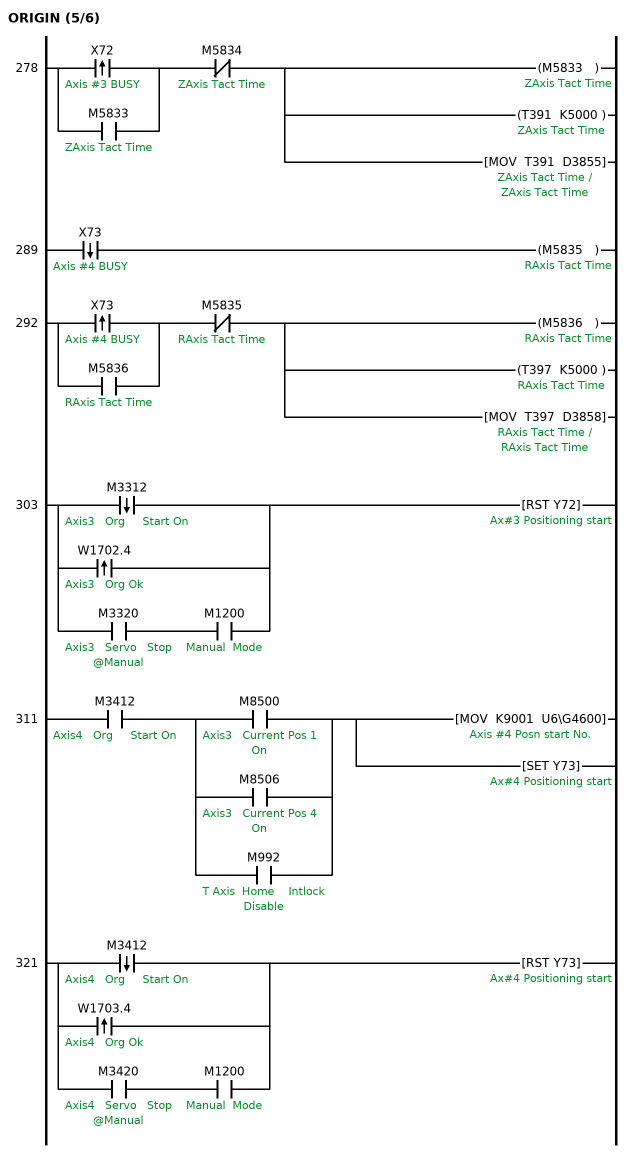
[picture p24: ladder of ORIGIN, rungs at steps 278 to 321]
278   LDP     X72  ; Axis #3 BUSY
      OR      M5833  ; ZAxis Tact Time
      ANI     M5834  ; ZAxis Tact Time
      OUT     M5833  ; ZAxis Tact Time
      OUT     T391 K5000  ; ZAxis Tact Time
      MOV     T391 D3855  ; ZAxis Tact Time
289   LDF     X73  ; Axis #4 BUSY
      OUT     M5835  ; RAxis Tact Time
292   LDP     X73  ; Axis #4 BUSY
      OR      M5836  ; RAxis Tact Time
      ANI     M5835  ; RAxis Tact Time
      OUT     M5836  ; RAxis Tact Time
      OUT     T397 K5000  ; RAxis Tact Time
      MOV     T397 D3858  ; RAxis Tact Time
303   LDF     M3312  ; Axis3   Org     Start On
      ORP     W1702.4  ; Axis3   Org Ok
      LD      M3320  ; Axis3   Servo   Stop    @Manual
      AND     M1200  ; Manual  Mode
      ORB
      RST     Y72  ; Ax#3 Positioning start
311   LD      M3412  ; Axis4   Org     Start On
      LD      M8500  ; Axis3   Current Pos 1 On
      OR      M8506  ; Axis3   Current Pos 4 On
      OR      M992  ; T Axis  Home    Intlock Disable
      ANB
      MOV     K9001 U6\G4600  ; Axis #4 Posn start No.
      SET     Y73  ; Ax#4 Positioning start
321   LDF     M3412  ; Axis4   Org     Start On
      ORP     W1703.4  ; Axis4   Org Ok
      LD      M3420  ; Axis4   Servo   Stop    @Manual
      AND     M1200  ; Manual  Mode
      ORB
      RST     Y73  ; Ax#4 Positioning start
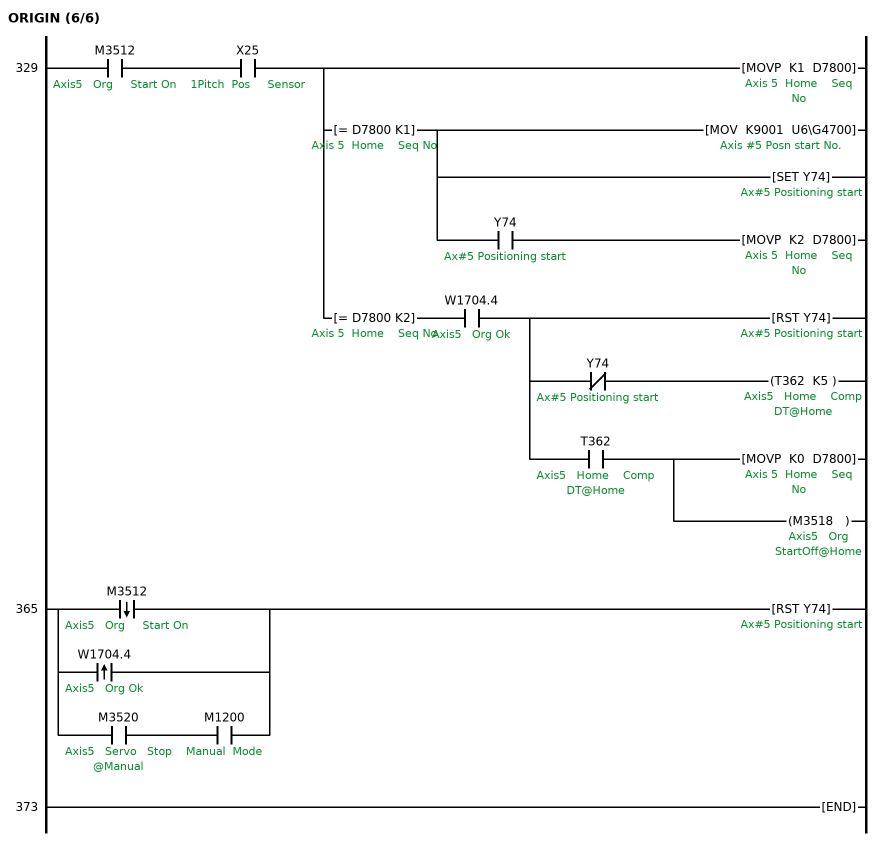
329   LD      M3512  ; Axis5   Org     Start On
      AND     X25  ; 1Pitch  Pos     Sensor
      MOVP    K1 D7800  ; Axis 5  Home    Seq No
      MPS
      AND=    D7800 K1  ; Axis 5  Home    Seq No
      MOV     K9001 U6\G4700  ; Axis #5 Posn start No.
      SET     Y74  ; Ax#5 Positioning start
      AND     Y74  ; Ax#5 Positioning start
      MOVP    K2 D7800
      MPP
      AND=    D7800 K2  ; Axis 5  Home    Seq No
      AND     W1704.4  ; Axis5   Org Ok
      RST     Y74  ; Ax#5 Positioning start
      MPS
      ANI     Y74  ; Ax#5 Positioning start
      OUT     T362 K5  ; Axis5   Home    Comp    DT@Home
      MPP
      AND     T362  ; Axis5   Home    Comp    DT@Home
      MOVP    K0 D7800
      OUT     M3518  ; Axis5   Org     StartOff@Home
365   LDF     M3512  ; Axis5   Org     Start On
      ORP     W1704.4  ; Axis5   Org Ok
      LD      M3520  ; Axis5   Servo   Stop    @Manual
      AND     M1200  ; Manual  Mode
      ORB
      RST     Y74  ; Ax#5 Positioning start
373   END
END_PROGRAM

PROGRAM ALARM
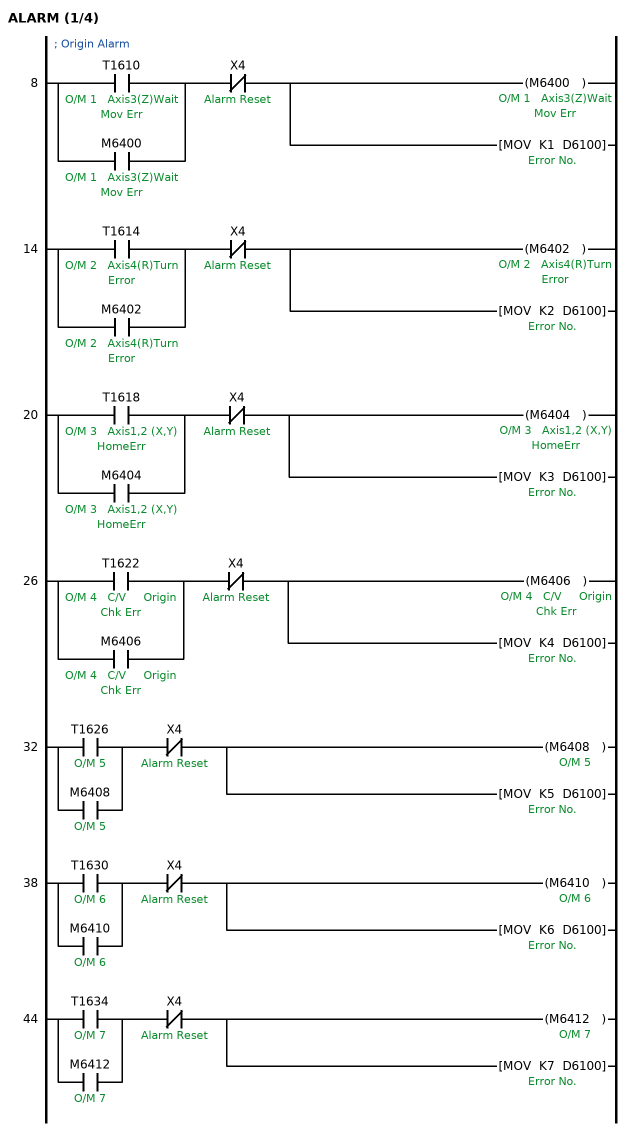
; Origin Alarm
8     LD      T1610  ; O/M 1   Axis3(Z)Wait    Mov Err
      OR      M6400  ; O/M 1   Axis3(Z)Wait    Mov Err
      ANI     X4  ; Alarm Reset
      OUT     M6400  ; O/M 1   Axis3(Z)Wait    Mov Err
      MOV     K1 D6100  ; Error No.
14    LD      T1614  ; O/M 2   Axis4(R)Turn    Error
      OR      M6402  ; O/M 2   Axis4(R)Turn    Error
      ANI     X4  ; Alarm Reset
      OUT     M6402  ; O/M 2   Axis4(R)Turn    Error
      MOV     K2 D6100
20    LD      T1618  ; O/M 3   Axis1,2 (X,Y)   HomeErr
      OR      M6404  ; O/M 3   Axis1,2 (X,Y)   HomeErr
      ANI     X4  ; Alarm Reset
      OUT     M6404  ; O/M 3   Axis1,2 (X,Y)   HomeErr
      MOV     K3 D6100
26    LD      T1622  ; O/M 4   C/V     Origin  Chk Err
      OR      M6406  ; O/M 4   C/V     Origin  Chk Err
      ANI     X4  ; Alarm Reset
      OUT     M6406  ; O/M 4   C/V     Origin  Chk Err
      MOV     K4 D6100
32    LD      T1626  ; O/M 5
      OR      M6408  ; O/M 5
      ANI     X4  ; Alarm Reset
      OUT     M6408  ; O/M 5
      MOV     K5 D6100
38    LD      T1630  ; O/M 6
      OR      M6410  ; O/M 6
      ANI     X4  ; Alarm Reset
      OUT     M6410  ; O/M 6
      MOV     K6 D6100
44    LD      T1634  ; O/M 7
      OR      M6412  ; O/M 7
      ANI     X4  ; Alarm Reset
      OUT     M6412  ; O/M 7
      MOV     K7 D6100
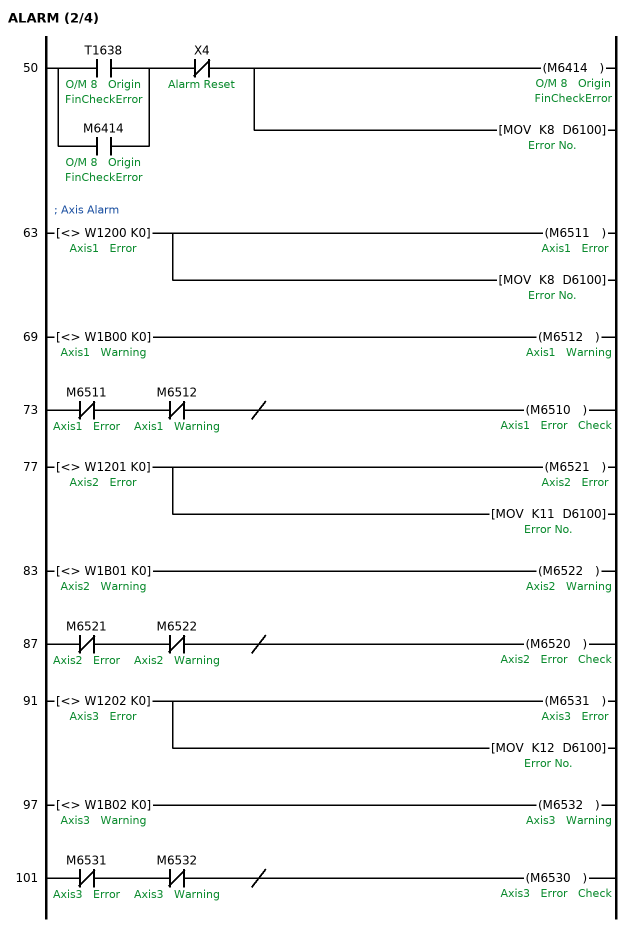
50    LD      T1638  ; O/M 8   Origin  FinCheckError
      OR      M6414  ; O/M 8   Origin  FinCheckError
      ANI     X4  ; Alarm Reset
      OUT     M6414  ; O/M 8   Origin  FinCheckError
      MOV     K8 D6100
; Axis Alarm
63    LD<>    W1200 K0  ; Axis1   Error
      OUT     M6511  ; Axis1   Error
      MOV     K8 D6100
69    LD<>    W1B00 K0  ; Axis1   Warning
      OUT     M6512  ; Axis1   Warning
73    LDI     M6511  ; Axis1   Error
      ANI     M6512  ; Axis1   Warning
      INV
      OUT     M6510  ; Axis1   Error   Check
77    LD<>    W1201 K0  ; Axis2   Error
      OUT     M6521  ; Axis2   Error
      MOV     K11 D6100
83    LD<>    W1B01 K0  ; Axis2   Warning
      OUT     M6522  ; Axis2   Warning
87    LDI     M6521  ; Axis2   Error
      ANI     M6522  ; Axis2   Warning
      INV
      OUT     M6520  ; Axis2   Error   Check
91    LD<>    W1202 K0  ; Axis3   Error
      OUT     M6531  ; Axis3   Error
      MOV     K12 D6100
97    LD<>    W1B02 K0  ; Axis3   Warning
      OUT     M6532  ; Axis3   Warning
101   LDI     M6531  ; Axis3   Error
      ANI     M6532  ; Axis3   Warning
      INV
      OUT     M6530  ; Axis3   Error   Check
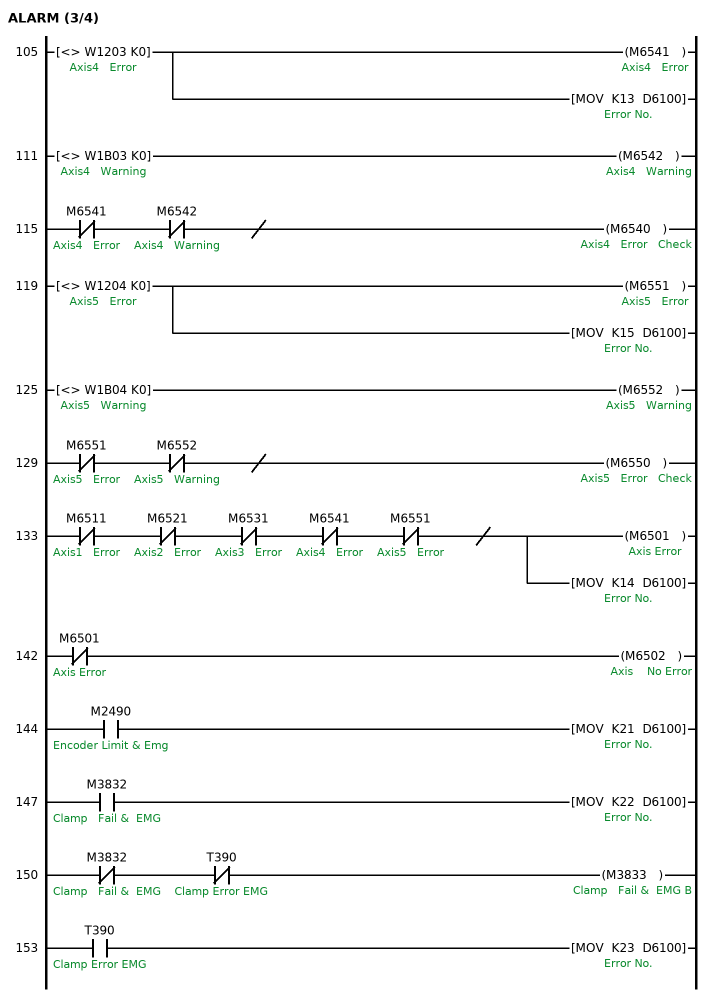
105   LD<>    W1203 K0  ; Axis4   Error
      OUT     M6541  ; Axis4   Error
      MOV     K13 D6100
111   LD<>    W1B03 K0  ; Axis4   Warning
      OUT     M6542  ; Axis4   Warning
115   LDI     M6541  ; Axis4   Error
      ANI     M6542  ; Axis4   Warning
      INV
      OUT     M6540  ; Axis4   Error   Check
119   LD<>    W1204 K0  ; Axis5   Error
      OUT     M6551  ; Axis5   Error
      MOV     K15 D6100
125   LD<>    W1B04 K0  ; Axis5   Warning
      OUT     M6552  ; Axis5   Warning
129   LDI     M6551  ; Axis5   Error
      ANI     M6552  ; Axis5   Warning
      INV
      OUT     M6550  ; Axis5   Error   Check
133   LDI     M6511  ; Axis1   Error
      ANI     M6521  ; Axis2   Error
      ANI     M6531  ; Axis3   Error
      ANI     M6541  ; Axis4   Error
      ANI     M6551  ; Axis5   Error
      INV
      OUT     M6501  ; Axis Error
      MOV     K14 D6100
142   LDI     M6501  ; Axis Error
      OUT     M6502  ; Axis    No Error
144   LD      M2490  ; Encoder Limit & Emg
      MOV     K21 D6100
147   LD      M3832  ; Clamp   Fail &  EMG
      MOV     K22 D6100
150   LDI     M3832  ; Clamp   Fail &  EMG
      ANI     T390  ; Clamp Error EMG
      OUT     M3833  ; Clamp   Fail &  EMG B
153   LD      T390  ; Clamp Error EMG
      MOV     K23 D6100
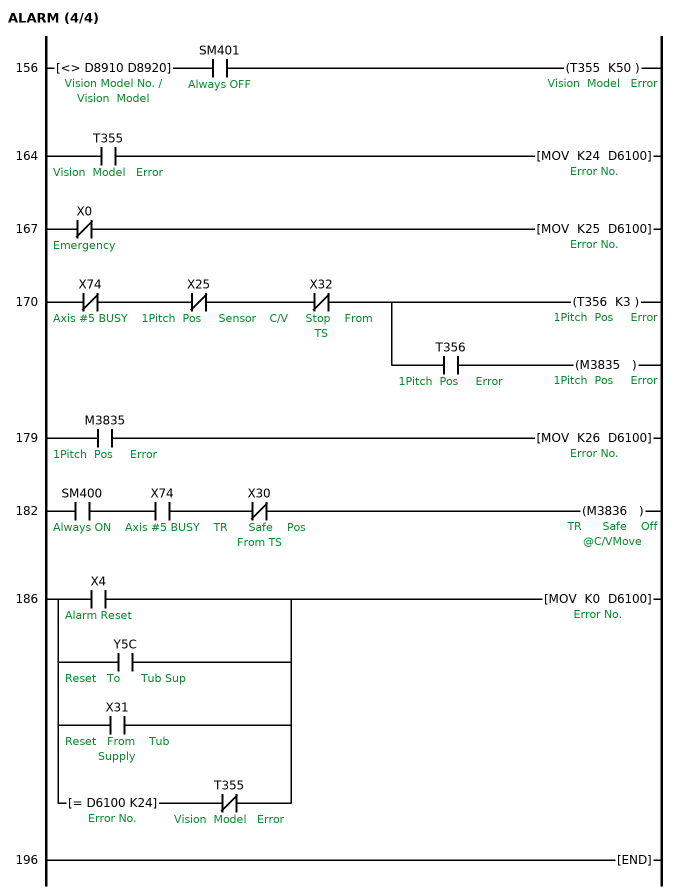
156   LD<>    D8910 D8920  ; Vision Model No. / Vision  Model
      AND     SM401  ; Always OFF
      OUT     T355 K50  ; Vision  Model   Error
164   LD      T355  ; Vision  Model   Error
      MOV     K24 D6100
167   LDI     X0  ; Emergency
      MOV     K25 D6100
170   LDI     X74  ; Axis #5 BUSY
      ANI     X25  ; 1Pitch  Pos     Sensor
      ANI     X32  ; C/V     Stop    From    TS
      OUT     T356 K3  ; 1Pitch  Pos     Error
      AND     T356  ; 1Pitch  Pos     Error
      OUT     M3835  ; 1Pitch  Pos     Error
179   LD      M3835  ; 1Pitch  Pos     Error
      MOV     K26 D6100
182   LD      SM400  ; Always ON
      AND     X74  ; Axis #5 BUSY
      ANI     X30  ; TR      Safe    Pos     From TS
      OUT     M3836  ; TR      Safe    Off     @C/VMove
186   LD      X4  ; Alarm Reset
      OR      Y5C  ; Reset   To      Tub Sup
      OR      X31  ; Reset   From    Tub     Supply
      LD=     D6100 K24  ; Error No.
      ANI     T355  ; Vision  Model   Error
      ORB
      MOV     K0 D6100
196   END
END_PROGRAM

PROGRAM SERVO
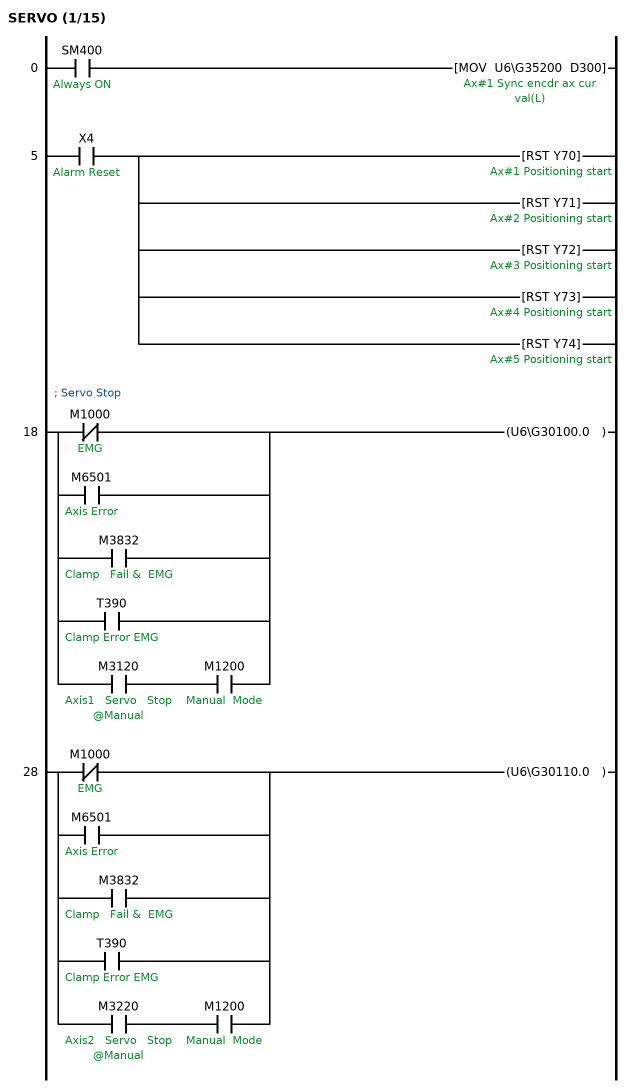
0     LD      SM400  ; Always ON
      MOV     U6\G35200 D300  ; Ax#1 Sync encdr ax cur val(L)
5     LD      X4  ; Alarm Reset
      RST     Y70  ; Ax#1 Positioning start
      RST     Y71  ; Ax#2 Positioning start
      RST     Y72  ; Ax#3 Positioning start
      RST     Y73  ; Ax#4 Positioning start
      RST     Y74  ; Ax#5 Positioning start
; Servo Stop
18    LDI     M1000  ; EMG
      OR      M6501  ; Axis Error
      OR      M3832  ; Clamp   Fail &  EMG
      OR      T390  ; Clamp Error EMG
      LD      M3120  ; Axis1   Servo   Stop    @Manual
      AND     M1200  ; Manual  Mode
      ORB
      OUT     U6\G30100.0
28    LDI     M1000  ; EMG
      OR      M6501  ; Axis Error
      OR      M3832  ; Clamp   Fail &  EMG
      OR      T390  ; Clamp Error EMG
      LD      M3220  ; Axis2   Servo   Stop    @Manual
      AND     M1200  ; Manual  Mode
      ORB
      OUT     U6\G30110.0
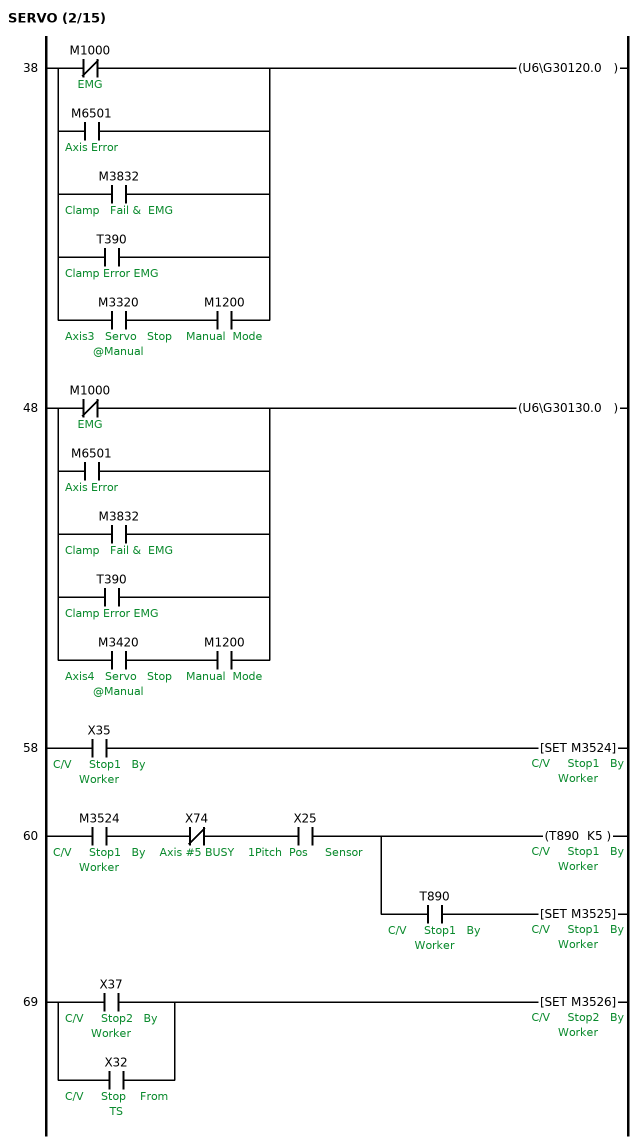
38    LDI     M1000  ; EMG
      OR      M6501  ; Axis Error
      OR      M3832  ; Clamp   Fail &  EMG
      OR      T390  ; Clamp Error EMG
      LD      M3320  ; Axis3   Servo   Stop    @Manual
      AND     M1200  ; Manual  Mode
      ORB
      OUT     U6\G30120.0
48    LDI     M1000  ; EMG
      OR      M6501  ; Axis Error
      OR      M3832  ; Clamp   Fail &  EMG
      OR      T390  ; Clamp Error EMG
      LD      M3420  ; Axis4   Servo   Stop    @Manual
      AND     M1200  ; Manual  Mode
      ORB
      OUT     U6\G30130.0
58    LD      X35  ; C/V     Stop1   By      Worker
      SET     M3524  ; C/V     Stop1   By      Worker
60    LD      M3524  ; C/V     Stop1   By      Worker
      ANI     X74  ; Axis #5 BUSY
      AND     X25  ; 1Pitch  Pos     Sensor
      OUT     T890 K5  ; C/V     Stop1   By      Worker
      AND     T890  ; C/V     Stop1   By      Worker
      SET     M3525  ; C/V     Stop1   By      Worker
69    LD      X37  ; C/V     Stop2   By      Worker
      OR      X32  ; C/V     Stop    From    TS
      SET     M3526  ; C/V     Stop2   By      Worker
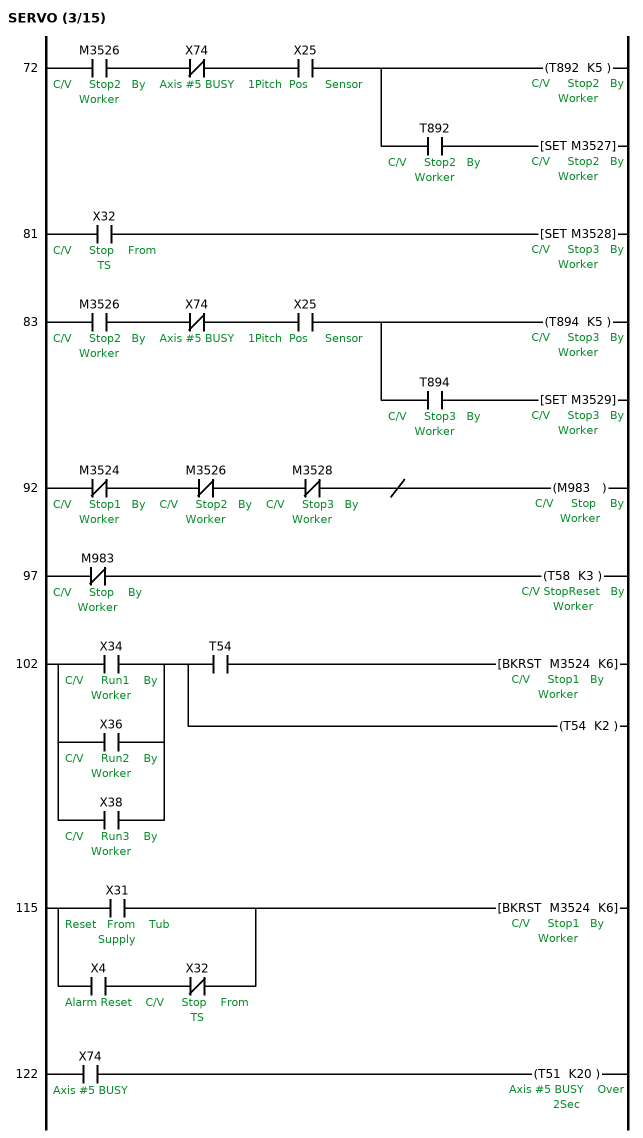
72    LD      M3526  ; C/V     Stop2   By      Worker
      ANI     X74  ; Axis #5 BUSY
      AND     X25  ; 1Pitch  Pos     Sensor
      OUT     T892 K5  ; C/V     Stop2   By      Worker
      AND     T892  ; C/V     Stop2   By      Worker
      SET     M3527  ; C/V     Stop2   By      Worker
81    LD      X32  ; C/V     Stop    From    TS
      SET     M3528  ; C/V     Stop3   By      Worker
83    LD      M3526  ; C/V     Stop2   By      Worker
      ANI     X74  ; Axis #5 BUSY
      AND     X25  ; 1Pitch  Pos     Sensor
      OUT     T894 K5  ; C/V     Stop3   By      Worker
      AND     T894  ; C/V     Stop3   By      Worker
      SET     M3529  ; C/V     Stop3   By      Worker
92    LDI     M3524  ; C/V     Stop1   By      Worker
      ANI     M3526  ; C/V     Stop2   By      Worker
      ANI     M3528  ; C/V     Stop3   By      Worker
      INV
      OUT     M983  ; C/V     Stop    By      Worker
97    LDI     M983  ; C/V     Stop    By      Worker
      OUT     T58 K3  ; C/V StopReset   By      Worker
102   LD      X34  ; C/V     Run1    By      Worker
      OR      X36  ; C/V     Run2    By      Worker
      OR      X38  ; C/V     Run3    By      Worker
      MPS
      AND     T54
      BKRST   M3524 K6
      MPP
      OUT     T54 K2
115   LD      X31  ; Reset   From    Tub     Supply
      LD      X4  ; Alarm Reset
      ANI     X32  ; C/V     Stop    From    TS
      ORB
      BKRST   M3524 K6
122   LD      X74  ; Axis #5 BUSY
      OUT     T51 K20  ; Axis #5 BUSY    Over    2Sec
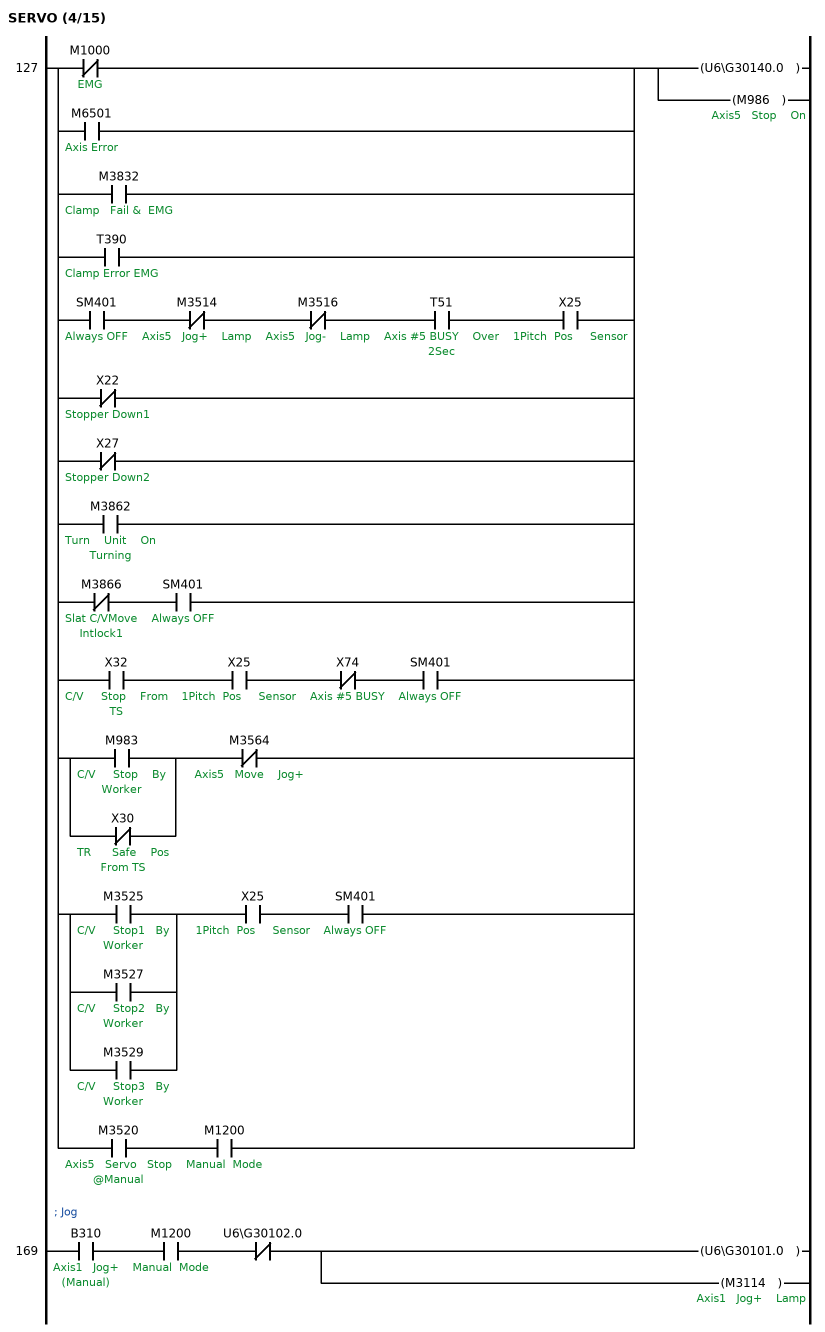
127   LDI     M1000  ; EMG
      OR      M6501  ; Axis Error
      OR      M3832  ; Clamp   Fail &  EMG
      OR      T390  ; Clamp Error EMG
      LD      SM401  ; Always OFF
      ANI     M3514  ; Axis5   Jog+    Lamp
      ANI     M3516  ; Axis5   Jog-    Lamp
      AND     T51  ; Axis #5 BUSY    Over    2Sec
      AND     X25  ; 1Pitch  Pos     Sensor
      ORB
      ORI     X22  ; Stopper Down1
      ORI     X27  ; Stopper Down2
      OR      M3862  ; Turn    Unit    On      Turning
      LDI     M3866  ; Slat C/VMove    Intlock1
      AND     SM401  ; Always OFF
      ORB
      LD      X32  ; C/V     Stop    From    TS
      AND     X25  ; 1Pitch  Pos     Sensor
      ANI     X74  ; Axis #5 BUSY
      AND     SM401  ; Always OFF
      ORB
      LD      M983  ; C/V     Stop    By      Worker
      ORI     X30  ; TR      Safe    Pos     From TS
      ANI     M3564  ; Axis5   Move    Jog+
      ORB
      LD      M3525  ; C/V     Stop1   By      Worker
      OR      M3527  ; C/V     Stop2   By      Worker
      OR      M3529  ; C/V     Stop3   By      Worker
      AND     X25  ; 1Pitch  Pos     Sensor
      AND     SM401  ; Always OFF
      ORB
      LD      M3520  ; Axis5   Servo   Stop    @Manual
      AND     M1200  ; Manual  Mode
      ORB
      OUT     U6\G30140.0
      OUT     M986  ; Axis5   Stop    On
; Jog
169   LD      B310  ; Axis1   Jog+    (Manual)
      AND     M1200  ; Manual  Mode
      ANI     U6\G30102.0
      OUT     U6\G30101.0
      OUT     M3114  ; Axis1   Jog+    Lamp
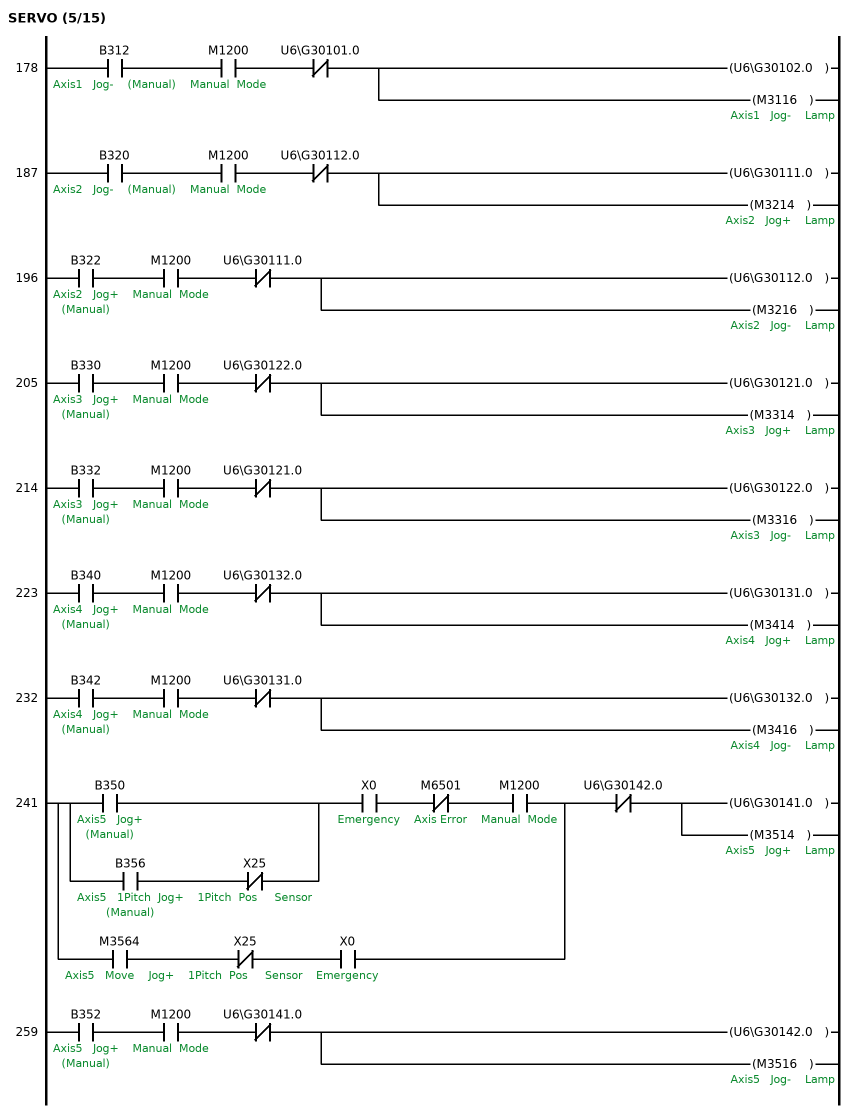
178   LD      B312  ; Axis1   Jog-    (Manual)
      AND     M1200  ; Manual  Mode
      ANI     U6\G30101.0
      OUT     U6\G30102.0
      OUT     M3116  ; Axis1   Jog-    Lamp
187   LD      B320  ; Axis2   Jog-    (Manual)
      AND     M1200  ; Manual  Mode
      ANI     U6\G30112.0
      OUT     U6\G30111.0
      OUT     M3214  ; Axis2   Jog+    Lamp
196   LD      B322  ; Axis2   Jog+    (Manual)
      AND     M1200  ; Manual  Mode
      ANI     U6\G30111.0
      OUT     U6\G30112.0
      OUT     M3216  ; Axis2   Jog-    Lamp
205   LD      B330  ; Axis3   Jog+    (Manual)
      AND     M1200  ; Manual  Mode
      ANI     U6\G30122.0
      OUT     U6\G30121.0
      OUT     M3314  ; Axis3   Jog+    Lamp
214   LD      B332  ; Axis3   Jog+    (Manual)
      AND     M1200  ; Manual  Mode
      ANI     U6\G30121.0
      OUT     U6\G30122.0
      OUT     M3316  ; Axis3   Jog-    Lamp
223   LD      B340  ; Axis4   Jog+    (Manual)
      AND     M1200  ; Manual  Mode
      ANI     U6\G30132.0
      OUT     U6\G30131.0
      OUT     M3414  ; Axis4   Jog+    Lamp
232   LD      B342  ; Axis4   Jog+    (Manual)
      AND     M1200  ; Manual  Mode
      ANI     U6\G30131.0
      OUT     U6\G30132.0
      OUT     M3416  ; Axis4   Jog-    Lamp
241   LD      B350  ; Axis5   Jog+    (Manual)
      LD      B356  ; Axis5   1Pitch  Jog+    (Manual)
      ANI     X25  ; 1Pitch  Pos     Sensor
      ORB
      AND     X0  ; Emergency
      ANI     M6501  ; Axis Error
      AND     M1200  ; Manual  Mode
      LD      M3564  ; Axis5   Move    Jog+
      ANI     X25  ; 1Pitch  Pos     Sensor
      AND     X0  ; Emergency
      ORB
      ANI     U6\G30142.0
      OUT     U6\G30141.0
      OUT     M3514  ; Axis5   Jog+    Lamp
259   LD      B352  ; Axis5   Jog+    (Manual)
      AND     M1200  ; Manual  Mode
      ANI     U6\G30141.0
      OUT     U6\G30142.0
      OUT     M3516  ; Axis5   Jog-    Lamp
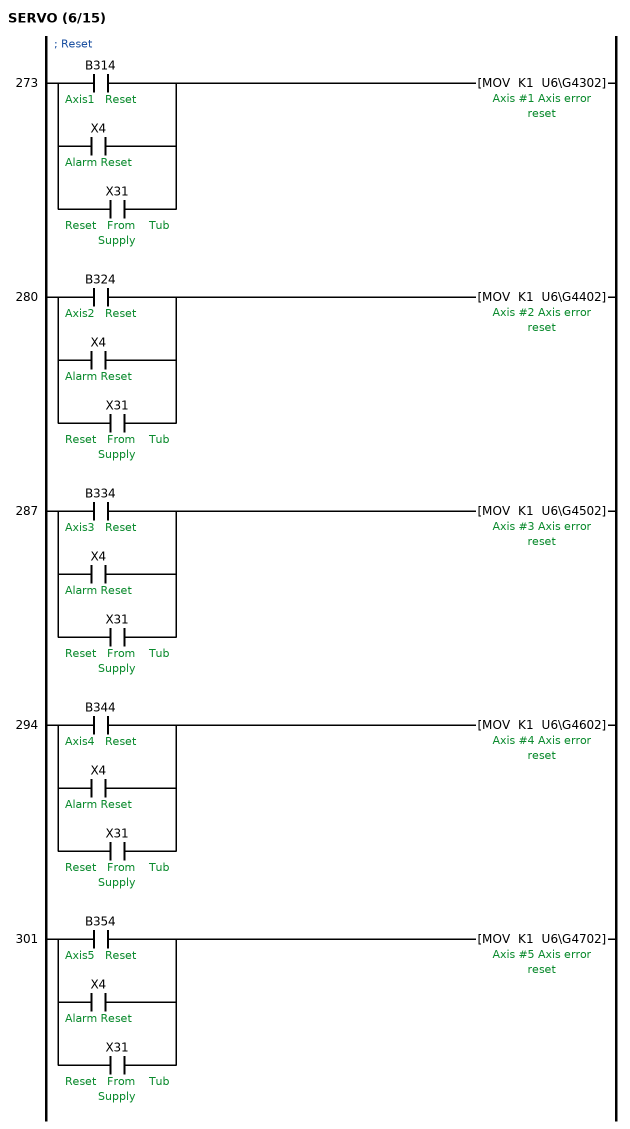
; Reset
273   LD      B314  ; Axis1   Reset
      OR      X4  ; Alarm Reset
      OR      X31  ; Reset   From    Tub     Supply
      MOV     K1 U6\G4302  ; Axis #1 Axis error reset
280   LD      B324  ; Axis2   Reset
      OR      X4  ; Alarm Reset
      OR      X31  ; Reset   From    Tub     Supply
      MOV     K1 U6\G4402  ; Axis #2 Axis error reset
287   LD      B334  ; Axis3   Reset
      OR      X4  ; Alarm Reset
      OR      X31  ; Reset   From    Tub     Supply
      MOV     K1 U6\G4502  ; Axis #3 Axis error reset
294   LD      B344  ; Axis4   Reset
      OR      X4  ; Alarm Reset
      OR      X31  ; Reset   From    Tub     Supply
      MOV     K1 U6\G4602  ; Axis #4 Axis error reset
301   LD      B354  ; Axis5   Reset
      OR      X4  ; Alarm Reset
      OR      X31  ; Reset   From    Tub     Supply
      MOV     K1 U6\G4702  ; Axis #5 Axis error reset
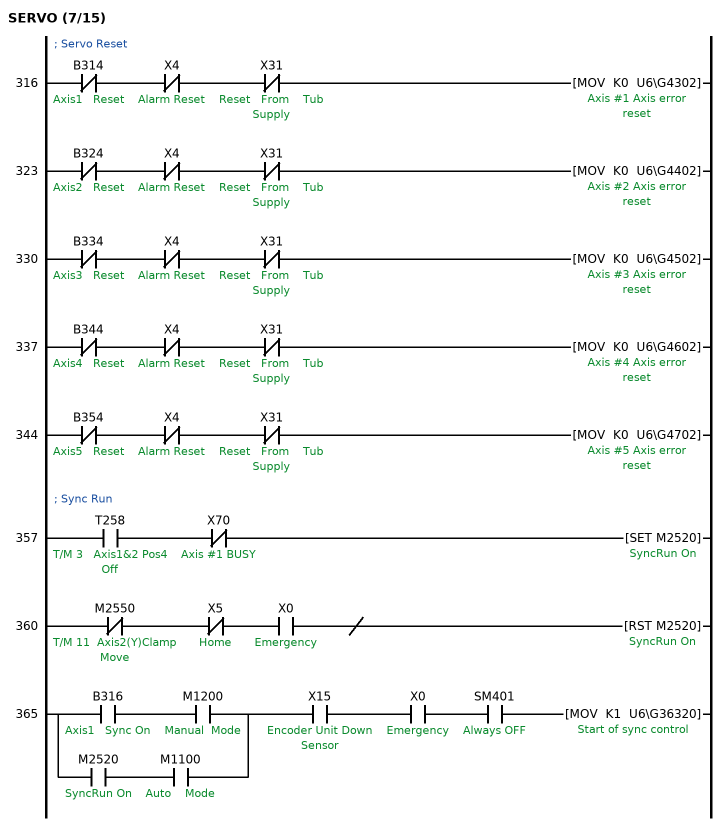
; Servo Reset
316   LDI     B314  ; Axis1   Reset
      ANI     X4  ; Alarm Reset
      ANI     X31  ; Reset   From    Tub     Supply
      MOV     K0 U6\G4302
323   LDI     B324  ; Axis2   Reset
      ANI     X4  ; Alarm Reset
      ANI     X31  ; Reset   From    Tub     Supply
      MOV     K0 U6\G4402
330   LDI     B334  ; Axis3   Reset
      ANI     X4  ; Alarm Reset
      ANI     X31  ; Reset   From    Tub     Supply
      MOV     K0 U6\G4502
337   LDI     B344  ; Axis4   Reset
      ANI     X4  ; Alarm Reset
      ANI     X31  ; Reset   From    Tub     Supply
      MOV     K0 U6\G4602
344   LDI     B354  ; Axis5   Reset
      ANI     X4  ; Alarm Reset
      ANI     X31  ; Reset   From    Tub     Supply
      MOV     K0 U6\G4702
; Sync Run
357   LD      T258  ; T/M 3   Axis1&2 Pos4    Off
      ANI     X70  ; Axis #1 BUSY
      SET     M2520  ; SyncRun On
360   LDI     M2550  ; T/M 11  Axis2(Y)Clamp   Move
      ANI     X5  ; Home
      AND     X0  ; Emergency
      INV
      RST     M2520  ; SyncRun On
365   LD      B316  ; Axis1   Sync On
      AND     M1200  ; Manual  Mode
      LD      M2520  ; SyncRun On
      AND     M1100  ; Auto    Mode
      ORB
      AND     X15  ; Encoder Unit Down Sensor
      AND     X0  ; Emergency
      AND     SM401  ; Always OFF
      MOV     K1 U6\G36320  ; Start of sync control
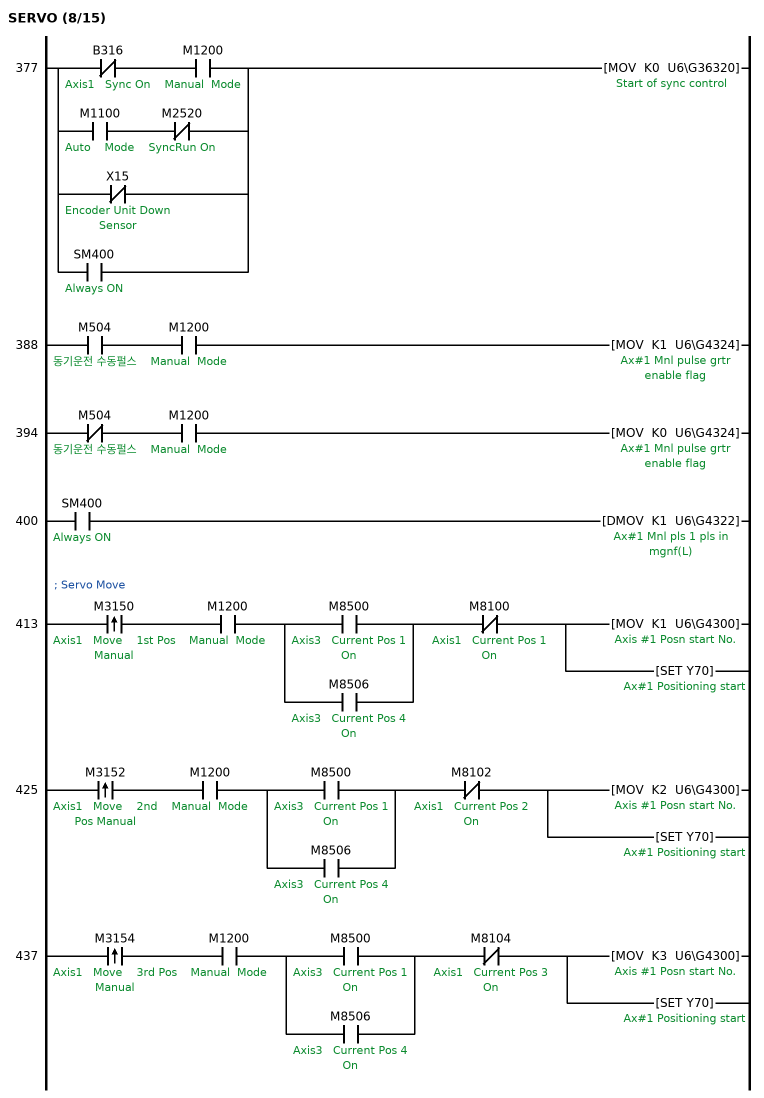
377   LDI     B316  ; Axis1   Sync On
      AND     M1200  ; Manual  Mode
      LD      M1100  ; Auto    Mode
      ANI     M2520  ; SyncRun On
      ORB
      ORI     X15  ; Encoder Unit Down Sensor
      OR      SM400  ; Always ON
      MOV     K0 U6\G36320
388   LD      M504  ; 동기운전 수동펄스
      AND     M1200  ; Manual  Mode
      MOV     K1 U6\G4324  ; Ax#1 Mnl pulse grtr enable flag
394   LDI     M504  ; 동기운전 수동펄스
      AND     M1200  ; Manual  Mode
      MOV     K0 U6\G4324
400   LD      SM400  ; Always ON
      DMOV    K1 U6\G4322  ; Ax#1 Mnl pls 1 pls in mgnf(L)
; Servo Move
413   LDP     M3150  ; Axis1   Move    1st Pos Manual
      AND     M1200  ; Manual  Mode
      LD      M8500  ; Axis3   Current Pos 1 On
      OR      M8506  ; Axis3   Current Pos 4 On
      ANB
      ANI     M8100  ; Axis1   Current Pos 1 On
      MOV     K1 U6\G4300  ; Axis #1 Posn start No.
      SET     Y70  ; Ax#1 Positioning start
425   LDP     M3152  ; Axis1   Move    2nd Pos Manual
      AND     M1200  ; Manual  Mode
      LD      M8500  ; Axis3   Current Pos 1 On
      OR      M8506  ; Axis3   Current Pos 4 On
      ANB
      ANI     M8102  ; Axis1   Current Pos 2 On
      MOV     K2 U6\G4300
      SET     Y70  ; Ax#1 Positioning start
437   LDP     M3154  ; Axis1   Move    3rd Pos Manual
      AND     M1200  ; Manual  Mode
      LD      M8500  ; Axis3   Current Pos 1 On
      OR      M8506  ; Axis3   Current Pos 4 On
      ANB
      ANI     M8104  ; Axis1   Current Pos 3 On
      MOV     K3 U6\G4300
      SET     Y70  ; Ax#1 Positioning start
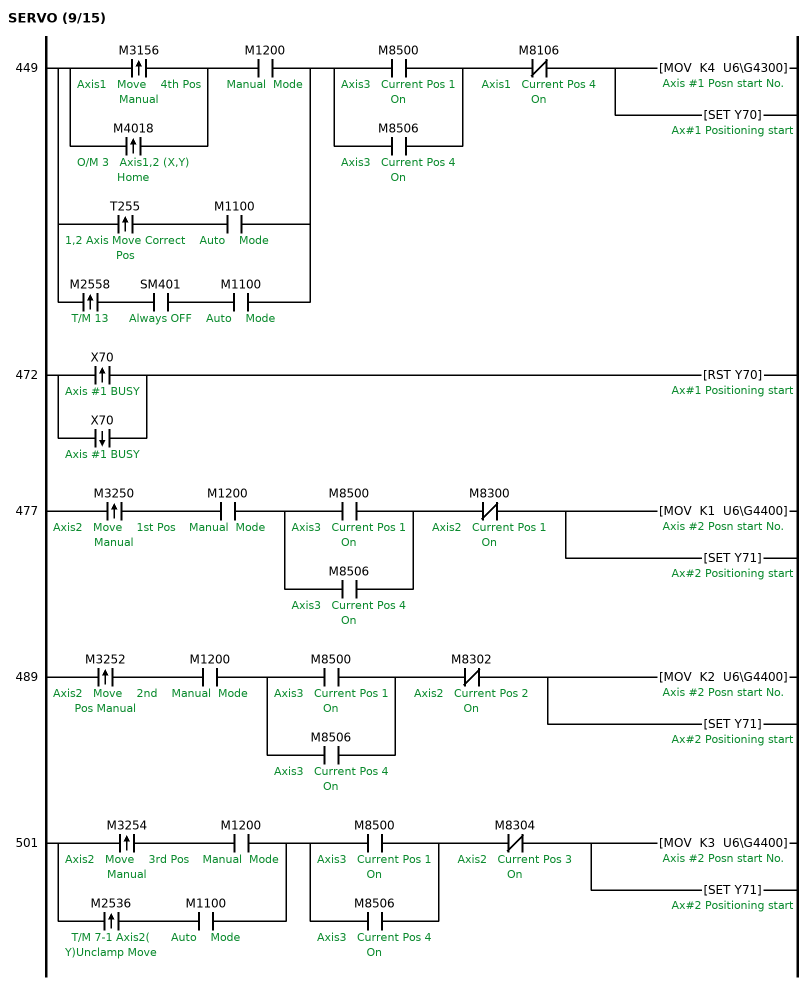
449   LDP     M3156  ; Axis1   Move    4th Pos Manual
      ORP     M4018  ; O/M 3   Axis1,2 (X,Y)   Home
      AND     M1200  ; Manual  Mode
      LDP     T255  ; 1,2 Axis Move Correct Pos
      AND     M1100  ; Auto    Mode
      ORB
      LDP     M2558  ; T/M 13
      AND     SM401  ; Always OFF
      AND     M1100  ; Auto    Mode
      ORB
      LD      M8500  ; Axis3   Current Pos 1 On
      OR      M8506  ; Axis3   Current Pos 4 On
      ANB
      ANI     M8106  ; Axis1   Current Pos 4 On
      MOV     K4 U6\G4300
      SET     Y70  ; Ax#1 Positioning start
472   LDP     X70  ; Axis #1 BUSY
      ORF     X70  ; Axis #1 BUSY
      RST     Y70  ; Ax#1 Positioning start
477   LDP     M3250  ; Axis2   Move    1st Pos Manual
      AND     M1200  ; Manual  Mode
      LD      M8500  ; Axis3   Current Pos 1 On
      OR      M8506  ; Axis3   Current Pos 4 On
      ANB
      ANI     M8300  ; Axis2   Current Pos 1 On
      MOV     K1 U6\G4400  ; Axis #2 Posn start No.
      SET     Y71  ; Ax#2 Positioning start
489   LDP     M3252  ; Axis2   Move    2nd Pos Manual
      AND     M1200  ; Manual  Mode
      LD      M8500  ; Axis3   Current Pos 1 On
      OR      M8506  ; Axis3   Current Pos 4 On
      ANB
      ANI     M8302  ; Axis2   Current Pos 2 On
      MOV     K2 U6\G4400
      SET     Y71  ; Ax#2 Positioning start
501   LDP     M3254  ; Axis2   Move    3rd Pos Manual
      AND     M1200  ; Manual  Mode
      LDP     M2536  ; T/M 7-1 Axis2(Y)Unclamp Move
      AND     M1100  ; Auto    Mode
      ORB
      LD      M8500  ; Axis3   Current Pos 1 On
      OR      M8506  ; Axis3   Current Pos 4 On
      ANB
      ANI     M8304  ; Axis2   Current Pos 3 On
      MOV     K3 U6\G4400
      SET     Y71  ; Ax#2 Positioning start
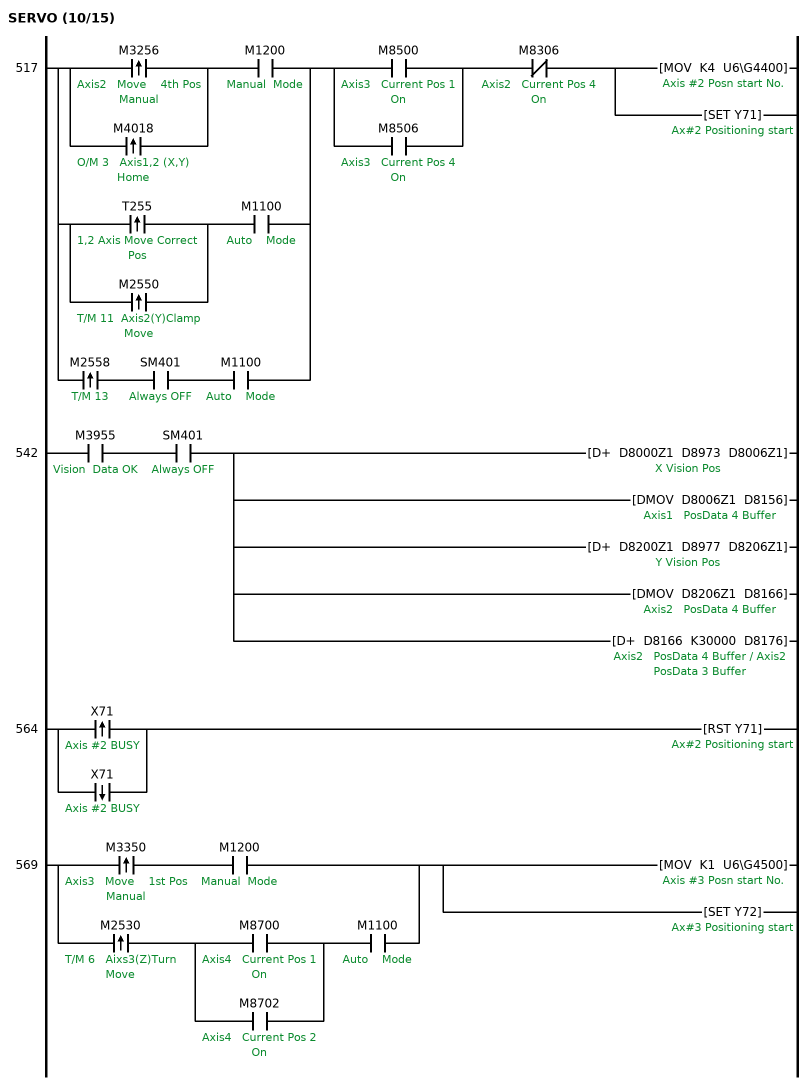
517   LDP     M3256  ; Axis2   Move    4th Pos Manual
      ORP     M4018  ; O/M 3   Axis1,2 (X,Y)   Home
      AND     M1200  ; Manual  Mode
      LDP     T255  ; 1,2 Axis Move Correct Pos
      ORP     M2550  ; T/M 11  Axis2(Y)Clamp   Move
      AND     M1100  ; Auto    Mode
      ORB
      LDP     M2558  ; T/M 13
      AND     SM401  ; Always OFF
      AND     M1100  ; Auto    Mode
      ORB
      LD      M8500  ; Axis3   Current Pos 1 On
      OR      M8506  ; Axis3   Current Pos 4 On
      ANB
      ANI     M8306  ; Axis2   Current Pos 4 On
      MOV     K4 U6\G4400
      SET     Y71  ; Ax#2 Positioning start
542   LD      M3955  ; Vision  Data OK
      AND     SM401  ; Always OFF
      D+      D8000Z1 D8973 D8006Z1  ; X Vision Pos
      DMOV    D8006Z1 D8156  ; Axis1   PosData 4 Buffer
      D+      D8200Z1 D8977 D8206Z1  ; Y Vision Pos
      DMOV    D8206Z1 D8166  ; Axis2   PosData 4 Buffer
      D+      D8166 K30000 D8176  ; Axis2   PosData 3 Buffer
564   LDP     X71  ; Axis #2 BUSY
      ORF     X71  ; Axis #2 BUSY
      RST     Y71  ; Ax#2 Positioning start
569   LDP     M3350  ; Axis3   Move    1st Pos Manual
      AND     M1200  ; Manual  Mode
      LDP     M2530  ; T/M 6   Aixs3(Z)Turn    Move
      LD      M8700  ; Axis4   Current Pos 1 On
      OR      M8702  ; Axis4   Current Pos 2 On
      ANB
      AND     M1100  ; Auto    Mode
      ORB
      MOV     K1 U6\G4500  ; Axis #3 Posn start No.
      SET     Y72  ; Ax#3 Positioning start
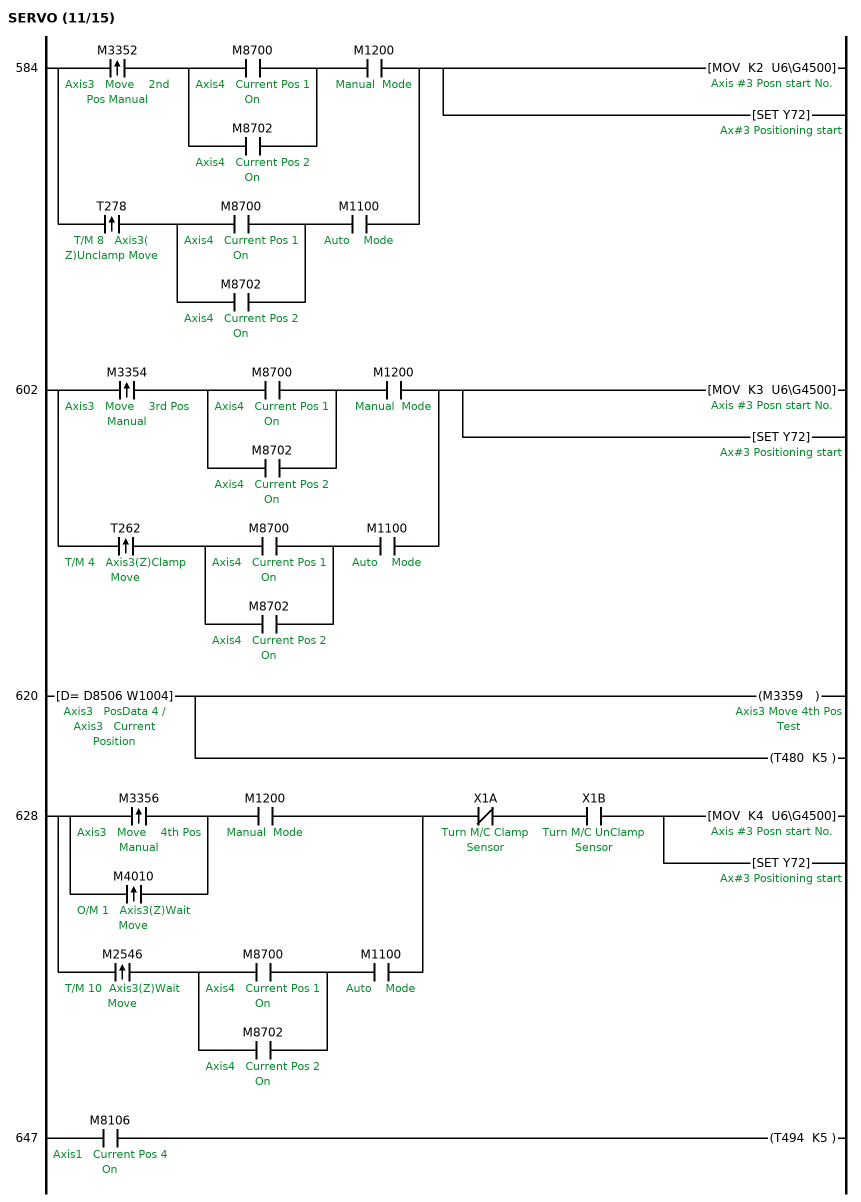
584   LDP     M3352  ; Axis3   Move    2nd Pos Manual
      LD      M8700  ; Axis4   Current Pos 1 On
      OR      M8702  ; Axis4   Current Pos 2 On
      ANB
      AND     M1200  ; Manual  Mode
      LDP     T278  ; T/M 8   Axis3(Z)Unclamp Move
      LD      M8700  ; Axis4   Current Pos 1 On
      OR      M8702  ; Axis4   Current Pos 2 On
      ANB
      AND     M1100  ; Auto    Mode
      ORB
      MOV     K2 U6\G4500
      SET     Y72  ; Ax#3 Positioning start
602   LDP     M3354  ; Axis3   Move    3rd Pos Manual
      LD      M8700  ; Axis4   Current Pos 1 On
      OR      M8702  ; Axis4   Current Pos 2 On
      ANB
      AND     M1200  ; Manual  Mode
      LDP     T262  ; T/M 4   Axis3(Z)Clamp   Move
      LD      M8700  ; Axis4   Current Pos 1 On
      OR      M8702  ; Axis4   Current Pos 2 On
      ANB
      AND     M1100  ; Auto    Mode
      ORB
      MOV     K3 U6\G4500
      SET     Y72  ; Ax#3 Positioning start
620   LDD=    D8506 W1004  ; Axis3   PosData 4 / Axis3   Current Position
      OUT     M3359  ; Axis3 Move 4th Pos Test
      OUT     T480 K5
628   LDP     M3356  ; Axis3   Move    4th Pos Manual
      ORP     M4010  ; O/M 1   Axis3(Z)Wait    Move
      AND     M1200  ; Manual  Mode
      LDP     M2546  ; T/M 10  Axis3(Z)Wait    Move
      LD      M8700  ; Axis4   Current Pos 1 On
      OR      M8702  ; Axis4   Current Pos 2 On
      ANB
      AND     M1100  ; Auto    Mode
      ORB
      ANI     X1A  ; Turn M/C Clamp Sensor
      AND     X1B  ; Turn M/C UnClamp Sensor
      MOV     K4 U6\G4500
      SET     Y72  ; Ax#3 Positioning start
647   LD      M8106  ; Axis1   Current Pos 4 On
      OUT     T494 K5
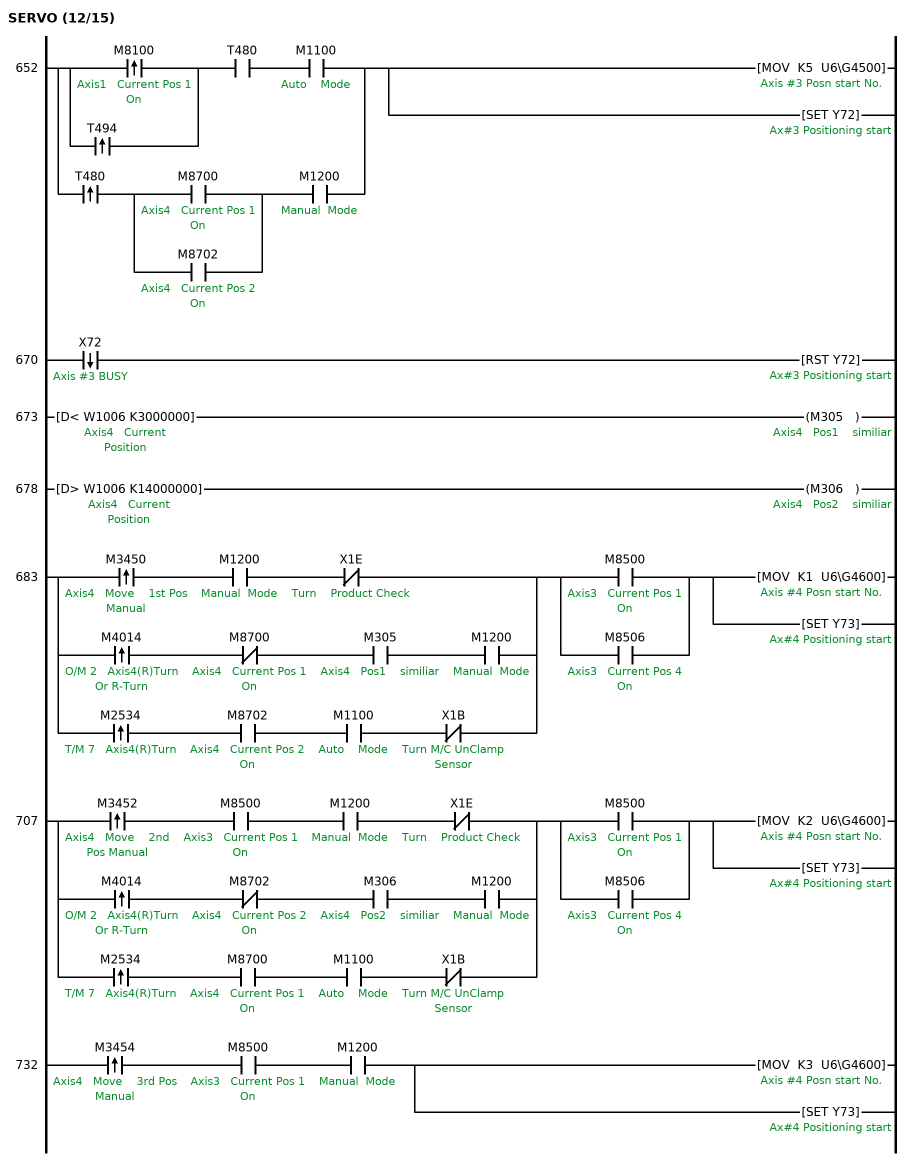
652   LDP     M8100  ; Axis1   Current Pos 1 On
      ORP     T494
      AND     T480
      AND     M1100  ; Auto    Mode
      LDP     T480
      LD      M8700  ; Axis4   Current Pos 1 On
      OR      M8702  ; Axis4   Current Pos 2 On
      ANB
      AND     M1200  ; Manual  Mode
      ORB
      MOV     K5 U6\G4500
      SET     Y72  ; Ax#3 Positioning start
670   LDF     X72  ; Axis #3 BUSY
      RST     Y72  ; Ax#3 Positioning start
673   LDD<    W1006 K3000000  ; Axis4   Current Position
      OUT     M305  ; Axis4   Pos1    similiar
678   LDD>    W1006 K14000000  ; Axis4   Current Position
      OUT     M306  ; Axis4   Pos2    similiar
683   LDP     M3450  ; Axis4   Move    1st Pos Manual
      AND     M1200  ; Manual  Mode
      ANI     X1E  ; Turn    Product Check
      LDP     M4014  ; O/M 2   Axis4(R)Turn Or R-Turn
      ANI     M8700  ; Axis4   Current Pos 1 On
      AND     M305  ; Axis4   Pos1    similiar
      AND     M1200  ; Manual  Mode
      ORB
      LDP     M2534  ; T/M 7   Axis4(R)Turn
      AND     M8702  ; Axis4   Current Pos 2 On
      AND     M1100  ; Auto    Mode
      ANI     X1B  ; Turn M/C UnClamp Sensor
      ORB
      LD      M8500  ; Axis3   Current Pos 1 On
      OR      M8506  ; Axis3   Current Pos 4 On
      ANB
      MOV     K1 U6\G4600  ; Axis #4 Posn start No.
      SET     Y73  ; Ax#4 Positioning start
707   LDP     M3452  ; Axis4   Move    2nd Pos Manual
      AND     M8500  ; Axis3   Current Pos 1 On
      AND     M1200  ; Manual  Mode
      ANI     X1E  ; Turn    Product Check
      LDP     M4014  ; O/M 2   Axis4(R)Turn Or R-Turn
      ANI     M8702  ; Axis4   Current Pos 2 On
      AND     M306  ; Axis4   Pos2    similiar
      AND     M1200  ; Manual  Mode
      ORB
      LDP     M2534  ; T/M 7   Axis4(R)Turn
      AND     M8700  ; Axis4   Current Pos 1 On
      AND     M1100  ; Auto    Mode
      ANI     X1B  ; Turn M/C UnClamp Sensor
      ORB
      LD      M8500  ; Axis3   Current Pos 1 On
      OR      M8506  ; Axis3   Current Pos 4 On
      ANB
      MOV     K2 U6\G4600
      SET     Y73  ; Ax#4 Positioning start
732   LDP     M3454  ; Axis4   Move    3rd Pos Manual
      AND     M8500  ; Axis3   Current Pos 1 On
      AND     M1200  ; Manual  Mode
      MOV     K3 U6\G4600
      SET     Y73  ; Ax#4 Positioning start
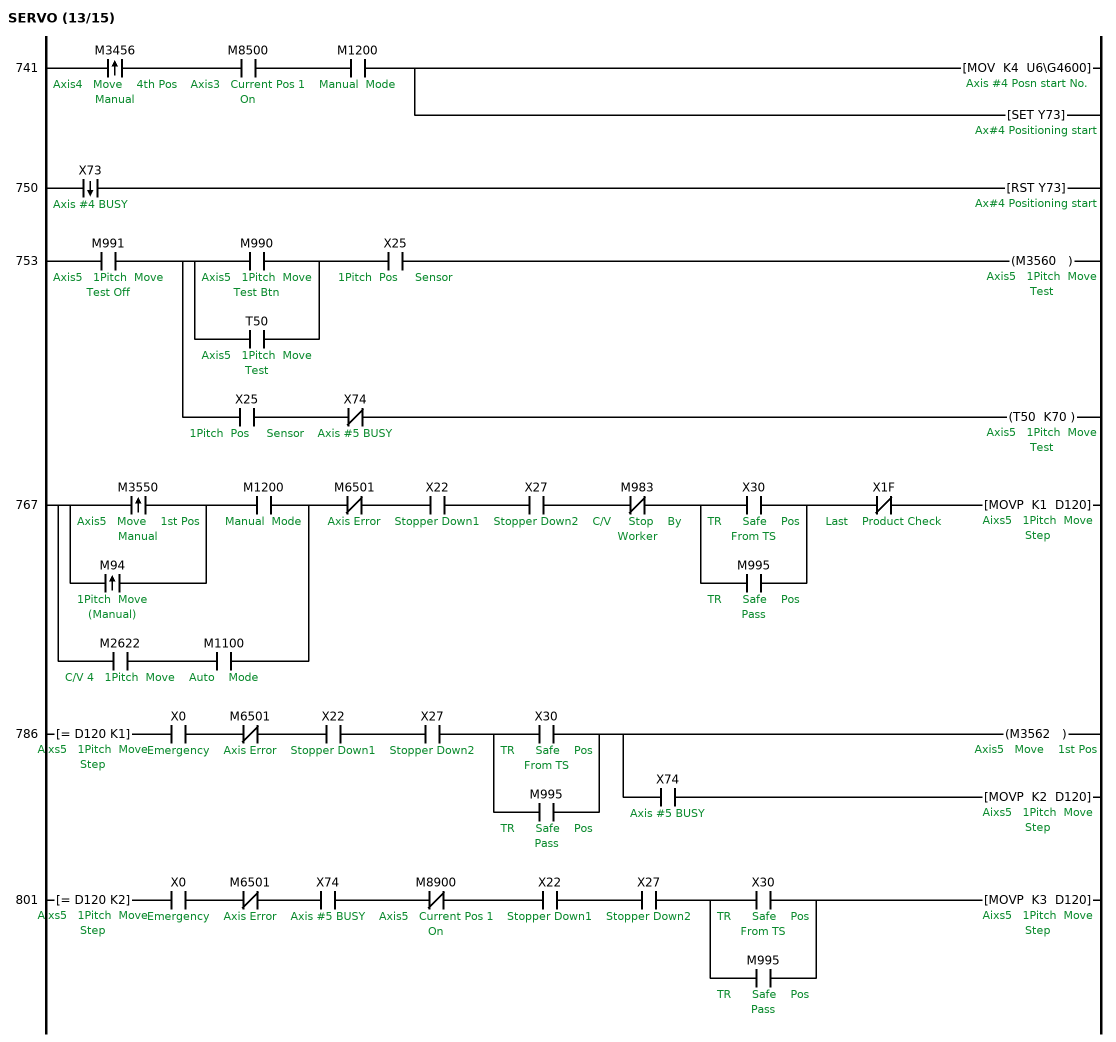
741   LDP     M3456  ; Axis4   Move    4th Pos Manual
      AND     M8500  ; Axis3   Current Pos 1 On
      AND     M1200  ; Manual  Mode
      MOV     K4 U6\G4600
      SET     Y73  ; Ax#4 Positioning start
750   LDF     X73  ; Axis #4 BUSY
      RST     Y73  ; Ax#4 Positioning start
753   LD      M991  ; Axis5   1Pitch  Move    Test Off
      MPS
      LD      M990  ; Axis5   1Pitch  Move    Test Btn
      OR      T50  ; Axis5   1Pitch  Move    Test
      ANB
      AND     X25  ; 1Pitch  Pos     Sensor
      OUT     M3560  ; Axis5   1Pitch  Move    Test
      MPP
      AND     X25  ; 1Pitch  Pos     Sensor
      ANI     X74  ; Axis #5 BUSY
      OUT     T50 K70  ; Axis5   1Pitch  Move    Test
767   LDP     M3550  ; Axis5   Move    1st Pos Manual
      ORP     M94  ; 1Pitch  Move    (Manual)
      AND     M1200  ; Manual  Mode
      LD      M2622  ; C/V 4   1Pitch  Move
      AND     M1100  ; Auto    Mode
      ORB
      ANI     M6501  ; Axis Error
      AND     X22  ; Stopper Down1
      AND     X27  ; Stopper Down2
      ANI     M983  ; C/V     Stop    By      Worker
      LD      X30  ; TR      Safe    Pos     From TS
      OR      M995  ; TR      Safe    Pos     Pass
      ANB
      ANI     X1F  ; Last    Product Check
      MOVP    K1 D120  ; Aixs5   1Pitch  Move    Step
786   LD=     D120 K1  ; Aixs5   1Pitch  Move    Step
      AND     X0  ; Emergency
      ANI     M6501  ; Axis Error
      AND     X22  ; Stopper Down1
      AND     X27  ; Stopper Down2
      LD      X30  ; TR      Safe    Pos     From TS
      OR      M995  ; TR      Safe    Pos     Pass
      ANB
      OUT     M3562  ; Axis5   Move    1st Pos
      AND     X74  ; Axis #5 BUSY
      MOVP    K2 D120
801   LD=     D120 K2  ; Aixs5   1Pitch  Move    Step
      AND     X0  ; Emergency
      ANI     M6501  ; Axis Error
      AND     X74  ; Axis #5 BUSY
      ANI     M8900  ; Axis5   Current Pos 1 On
      AND     X22  ; Stopper Down1
      AND     X27  ; Stopper Down2
      LD      X30  ; TR      Safe    Pos     From TS
      OR      M995  ; TR      Safe    Pos     Pass
      ANB
      MOVP    K3 D120
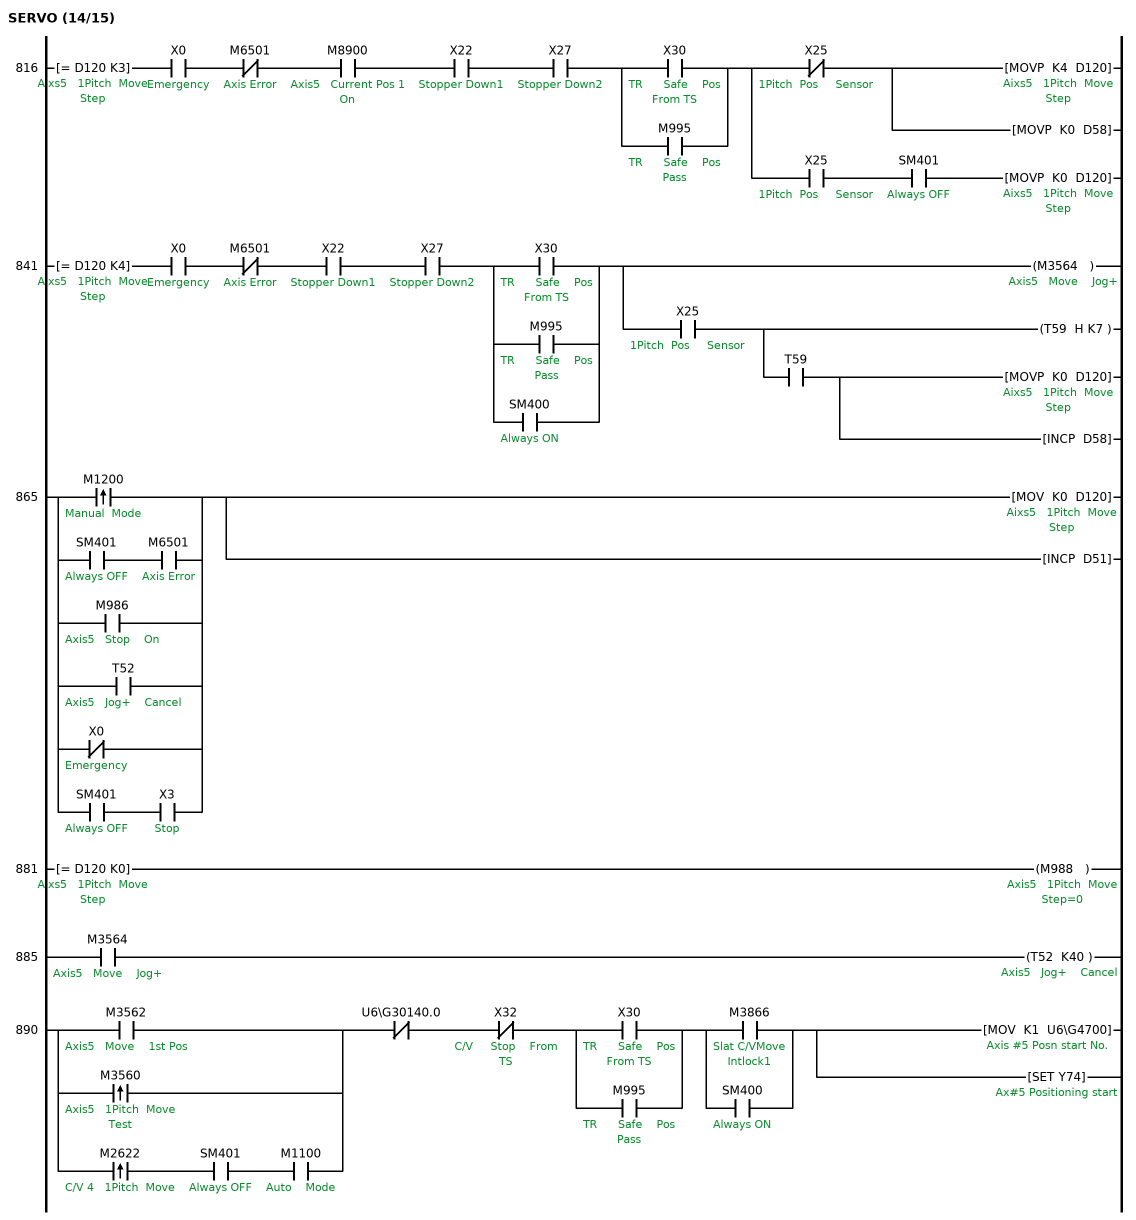
816   LD=     D120 K3  ; Aixs5   1Pitch  Move    Step
      AND     X0  ; Emergency
      ANI     M6501  ; Axis Error
      AND     M8900  ; Axis5   Current Pos 1 On
      AND     X22  ; Stopper Down1
      AND     X27  ; Stopper Down2
      LD      X30  ; TR      Safe    Pos     From TS
      OR      M995  ; TR      Safe    Pos     Pass
      ANB
      MPS
      ANI     X25  ; 1Pitch  Pos     Sensor
      MOVP    K4 D120
      MOVP    K0 D58
      MPP
      AND     X25  ; 1Pitch  Pos     Sensor
      AND     SM401  ; Always OFF
      MOVP    K0 D120
841   LD=     D120 K4  ; Aixs5   1Pitch  Move    Step
      AND     X0  ; Emergency
      ANI     M6501  ; Axis Error
      AND     X22  ; Stopper Down1
      AND     X27  ; Stopper Down2
      LD      X30  ; TR      Safe    Pos     From TS
      OR      M995  ; TR      Safe    Pos     Pass
      OR      SM400  ; Always ON
      ANB
      OUT     M3564  ; Axis5   Move    Jog+
      AND     X25  ; 1Pitch  Pos     Sensor
      OUTH    T59 K7
      AND     T59
      MOVP    K0 D120
      INCP    D58
865   LDP     M1200  ; Manual  Mode
      LD      SM401  ; Always OFF
      AND     M6501  ; Axis Error
      ORB
      OR      M986  ; Axis5   Stop    On
      OR      T52  ; Axis5   Jog+    Cancel
      ORI     X0  ; Emergency
      LD      SM401  ; Always OFF
      AND     X3  ; Stop
      ORB
      MOV     K0 D120
      INCP    D51
881   LD=     D120 K0  ; Aixs5   1Pitch  Move    Step
      OUT     M988  ; Axis5   1Pitch  Move    Step=0
885   LD      M3564  ; Axis5   Move    Jog+
      OUT     T52 K40  ; Axis5   Jog+    Cancel
890   LD      M3562  ; Axis5   Move    1st Pos
      ORP     M3560  ; Axis5   1Pitch  Move    Test
      LDP     M2622  ; C/V 4   1Pitch  Move
      AND     SM401  ; Always OFF
      AND     M1100  ; Auto    Mode
      ORB
      ANI     U6\G30140.0
      ANI     X32  ; C/V     Stop    From    TS
      LD      X30  ; TR      Safe    Pos     From TS
      OR      M995  ; TR      Safe    Pos     Pass
      ANB
      LD      M3866  ; Slat C/VMove    Intlock1
      OR      SM400  ; Always ON
      ANB
      MOV     K1 U6\G4700  ; Axis #5 Posn start No.
      SET     Y74  ; Ax#5 Positioning start
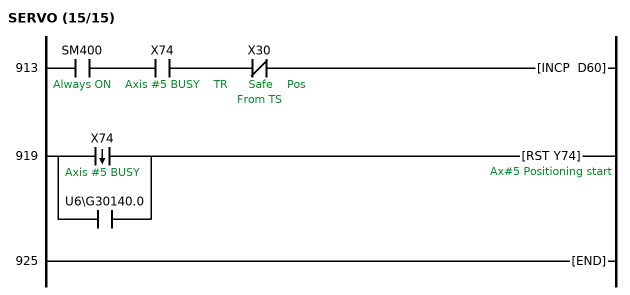
913   LD      SM400  ; Always ON
      AND     X74  ; Axis #5 BUSY
      ANI     X30  ; TR      Safe    Pos     From TS
      INCP    D60
919   LDF     X74  ; Axis #5 BUSY
      OR      U6\G30140.0
      RST     Y74  ; Ax#5 Positioning start
925   END
END_PROGRAM

PROGRAM DATA
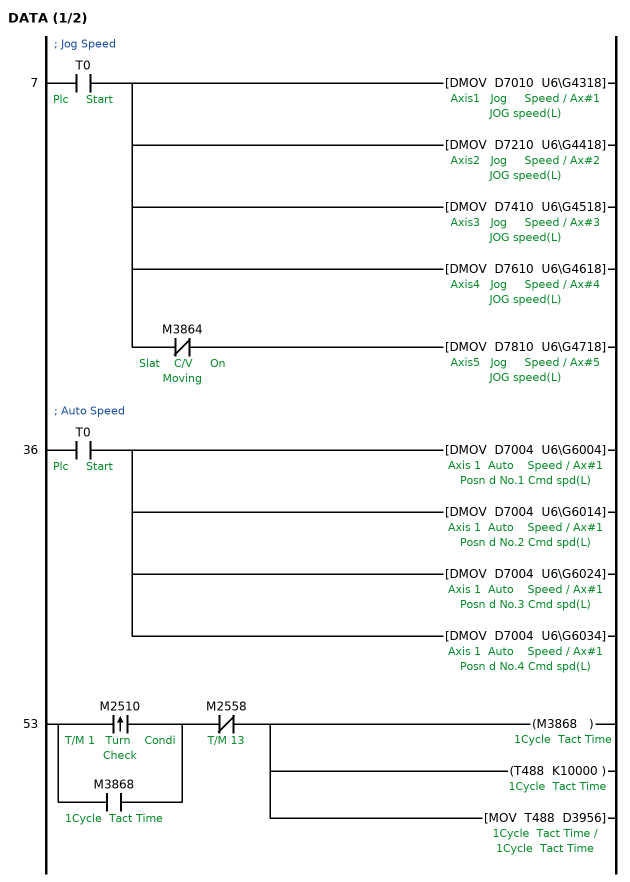
; Jog Speed
7     LD      T0  ; Plc     Start
      DMOV    D7010 U6\G4318  ; Axis1   Jog     Speed / Ax#1 JOG speed(L)
      DMOV    D7210 U6\G4418  ; Axis2   Jog     Speed / Ax#2 JOG speed(L)
      DMOV    D7410 U6\G4518  ; Axis3   Jog     Speed / Ax#3 JOG speed(L)
      DMOV    D7610 U6\G4618  ; Axis4   Jog     Speed / Ax#4 JOG speed(L)
      ANI     M3864  ; Slat    C/V     On      Moving
      DMOV    D7810 U6\G4718  ; Axis5   Jog     Speed / Ax#5 JOG speed(L)
; Auto Speed
36    LD      T0  ; Plc     Start
      DMOV    D7004 U6\G6004  ; Axis 1  Auto    Speed / Ax#1 Posn d No.1 Cmd spd(L)
      DMOV    D7004 U6\G6014  ; Ax#1 Posn d No.2 Cmd spd(L)
      DMOV    D7004 U6\G6024  ; Ax#1 Posn d No.3 Cmd spd(L)
      DMOV    D7004 U6\G6034  ; Ax#1 Posn d No.4 Cmd spd(L)
53    LDP     M2510  ; T/M 1   Turn    Condi   Check
      OR      M3868  ; 1Cycle  Tact Time
      ANI     M2558  ; T/M 13
      OUT     M3868  ; 1Cycle  Tact Time
      OUT     T488 K10000  ; 1Cycle  Tact Time
      MOV     T488 D3956  ; 1Cycle  Tact Time
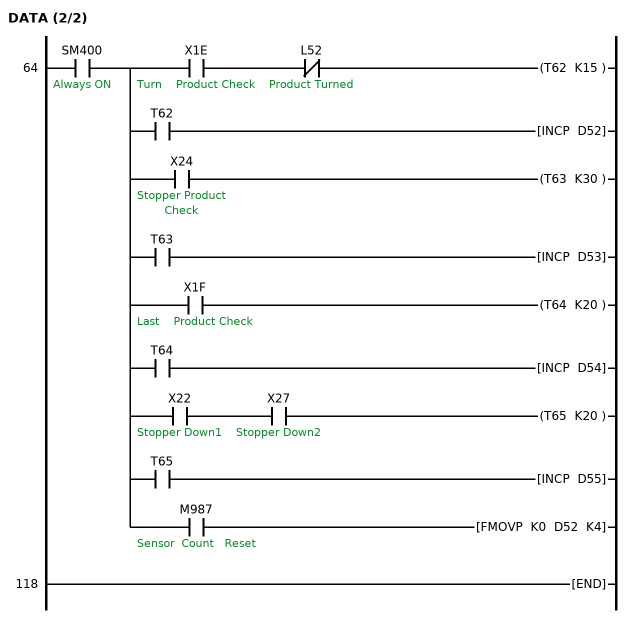
64    LD      SM400  ; Always ON
      MPS
      AND     X1E  ; Turn    Product Check
      ANI     L52  ; Product Turned
      OUT     T62 K15
      MRD
      AND     T62
      INCP    D52
      MRD
      AND     X24  ; Stopper Product Check
      OUT     T63 K30
      MRD
      AND     T63
      INCP    D53
      MRD
      AND     X1F  ; Last    Product Check
      OUT     T64 K20
      MRD
      AND     T64
      INCP    D54
      MRD
      AND     X22  ; Stopper Down1
      AND     X27  ; Stopper Down2
      OUT     T65 K20
      MRD
      AND     T65
      INCP    D55
      MPP
      AND     M987  ; Sensor  Count   Reset
      FMOVP   K0 D52 K4
118   END
END_PROGRAM

PROGRAM CONSTDAT
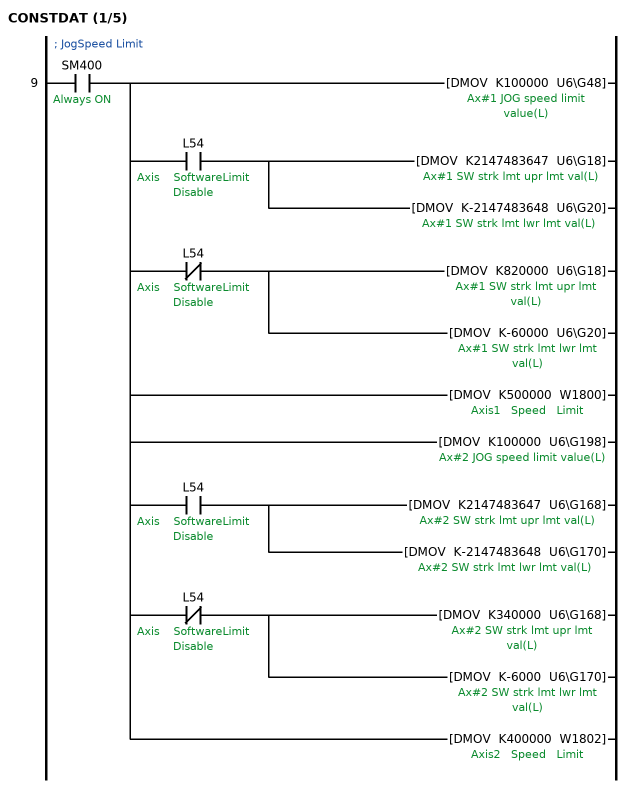
; JogSpeed Limit
9     LD      SM400  ; Always ON
      DMOV    K100000 U6\G48  ; Ax#1 JOG speed limit value(L)
      MPS
      AND     L54  ; Axis    SoftwareLimit   Disable
      DMOV    K2147483647 U6\G18  ; Ax#1 SW strk lmt upr lmt val(L)
      DMOV    K-2147483648 U6\G20  ; Ax#1 SW strk lmt lwr lmt val(L)
      MRD
      ANI     L54  ; Axis    SoftwareLimit   Disable
      DMOV    K820000 U6\G18
      DMOV    K-60000 U6\G20
      MPP
      DMOV    K500000 W1800  ; Axis1   Speed   Limit
      DMOV    K100000 U6\G198  ; Ax#2 JOG speed limit value(L)
      MPS
      AND     L54  ; Axis    SoftwareLimit   Disable
      DMOV    K2147483647 U6\G168  ; Ax#2 SW strk lmt upr lmt val(L)
      DMOV    K-2147483648 U6\G170  ; Ax#2 SW strk lmt lwr lmt val(L)
      MRD
      ANI     L54  ; Axis    SoftwareLimit   Disable
      DMOV    K340000 U6\G168
      DMOV    K-6000 U6\G170
      MPP
      DMOV    K400000 W1802  ; Axis2   Speed   Limit
